// TIA Portal V21 export
DATA_BLOCK "DiagnosticaProfinet"   // DB36
{ S7_Optimized_Access := 'TRUE' }
// stored: MemoryReserve 100
   VAR
      AllarmiRicercaDisp : Struct   // Allarmi dovuti alla ricerca dei dispositivi
         Configurati : String := 'Tutto ok';
         Disturbati : String := 'Tutto ok';
         Disattivati : String := 'Tutto ok';
         Disponibili : String := 'Tutto ok';
         ConWarning : String := 'Tutto ok';
      END_STRUCT;
      Dispositivo : Array[0.."K_NumDispositivoProfinet"] of Struct
         Configurato : Bool;
         Disturbato : Bool;
         Disattivato : Bool;
         Disponibile : Bool;
         SegnalazionePresente : Bool;
         Stato : Int;   // 0 = NonConfigurato 1=Configurato 2=Configurato&Disattivato 3=Configurato&SegnalazionePresente 4=Configurato&Disponibile 5=Configurato&Disturbato 6=Configurato&NonDisponibile
         WordHMI : Word;
      END_STRUCT;
   END_VAR
BEGIN
   Dispositivo[0].Configurato := TRUE;
   Dispositivo[0].Disturbato := FALSE;
   Dispositivo[0].Disattivato := FALSE;
   Dispositivo[0].Disponibile := TRUE;
   Dispositivo[0].SegnalazionePresente := FALSE;
   Dispositivo[0].Stato := 4;
   Dispositivo[0].WordHMI := 16#0000;
END_DATA_BLOCK
